FUNCTION_BLOCK DoorSensor (* Template for a simple Basic Function Block Type *)
  (* Standard: 61499-2 *)
  (* Version 1.0, 2019-05-09, jetbrains *)
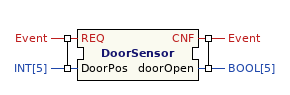
  EVENT_INPUT
    REQ WITH DoorPos; (* Normal Execution Request *)
  END_EVENT
  EVENT_OUTPUT
    CNF WITH doorOpen; (* Execution Confirmation *)
  END_EVENT
  VAR_INPUT
    DoorPos : ARRAY [0..4] OF INT; (* Input event qualifier *)
  END_VAR
  VAR_OUTPUT
    doorOpen : ARRAY [0..4] OF BOOL;
  END_VAR
  VAR
    prevPos : ARRAY [0..4] OF INT := -1; (* Internal Variable *)
  END_VAR
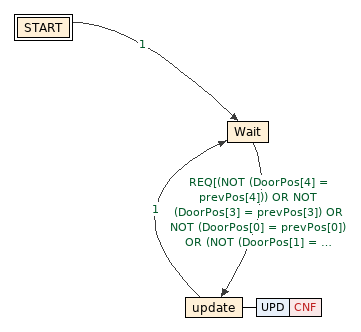
  EC_STATES
    START; (* Initial State *)
    update : UPD -> CNF;
    Wait;
  END_STATES
  EC_TRANSITIONS
    Wait TO update := REQ[(NOT (DoorPos[4] = prevPos[4])) OR  NOT (DoorPos[3] = prevPos[3]) OR  NOT (DoorPos[0] = prevPos[0]) OR (NOT (DoorPos[1] = prevPos[1])) OR (NOT (DoorPos[2] = prevPos[2]))];
    update TO Wait := 1;
    START TO Wait := 1;
  END_TRANSITIONS
  ALGORITHM initialize IN ST: (* Initialization algorithm *)
prevPos[0]  := DoorPos[0];
prevPos[1]  := DoorPos[1];
prevPos[2]  := DoorPos[2];
  END_ALGORITHM
  ALGORITHM UPD IN ST: (* new algorithm *)
doorOpen[0] := DoorPos[0] = 10;
doorOpen[1] := DoorPos[1] = 10;
doorOpen[2] := DoorPos[2] = 10;
doorOpen[3] := DoorPos[3] = 10;
doorOpen[4] := DoorPos[4] = 10;
prevPos[0] := DoorPos[0];
prevPos[1] := DoorPos[1];
prevPos[2] := DoorPos[2];
prevPos[3] := DoorPos[3];
prevPos[4] := DoorPos[4];
  END_ALGORITHM
END_FUNCTION_BLOCK
